# EPICS StreamDevice protocol: iocs/estherVacuumRpi/vacApp/Db/gate-valve.proto
Terminator = CR LF;
#Terminator = LF;
#LockTimeout = 5000;
ReplyTimeout = 2000;
#ReadTimeout  = 200;
#WriteTimeout = 100;
MaxInput     = 100;
#ExtraInput   = Error;
#ExtraInput   = Ignore;

#      "1, Closed, Char:x, SwIN:0, SwOUT:0, LimIN:1, LimOUT:0, Millis:1210605, Holding:1147167"

#1, Stopped, Char:x, SwIN:0, SwOUT:0, LimIN:0, LimOUT:0, Millis:686343, Holding:0
Millis {
    in "\$1, %*{Stopped|MovingIn|MovingOut|Closed|Open|Error}, Char:%*c, SwIN:%*b, SwOUT:%*b, LimIN:%*b, LimOUT:%*b, Millis:%d, Holding:%*d";
}
Box {
    in "%d, Closed, Char: x, SwIN: %*d, SwOUT: 0, LimIN: 1, LimOUT: 0, Millis: %*d,%*20c";
}
SwitchIn {
    in "\$1, %*{Stopped|MovingIn|MovingOut|Closed|Open|Error}, Char:%*c, SwIN:%b, SwOUT:%*b, LimIN:%*b, LimOUT:%*b, Millis:%*d, Holding:%*d";
}
SwitchInCmd {
    out "%{x|i|I}"
}

SwitchOut {
    in "\$1, %*{Stopped|MovingIn|MovingOut|Closed|Open|Error}, Char:%*c, SwIN:%*b, SwOUT:%b, LimIN:%*b, LimOUT:%*b, Millis:%*d, Holding:%*d";
}

SwitchOutCmd {
    out "%{x|o|O}"
}

StopCmd {
    out "s"
}

LimitIn {
    in "\$1, %*{Stopped|MovingIn|MovingOut|Closed|Open|Error}, Char:%*c, SwIN:%*b, SwOUT:%*b, LimIN:%b, LimOUT:%*b, Millis:%*d, Holding:%*d";
}

LimitOut {
    in "\$1, %*{Stopped|MovingIn|MovingOut|Closed|Open|Error}, Char:%*c, SwIN:%*b, SwOUT:%*b, LimIN:%*b, LimOUT:%b, Millis:%*d, Holding:%*d";
}

Status {
    in "\$1, %{Stopped|MovingIn|MovingOut|Closed|Open|Error}, Char:%*c, SwIN:%*b, SwOUT:%*b, LimIN:%*b, LimOUT:%*b, Millis:%*d, Holding:%*d";
}

    #in "\$1, %*{Stopped|MovingIn|MovingOut|Closed|Open|Error}, Char:%c, SwIN:%*b, SwOUT:%*b, LimIN:%*b, LimOUT:%*b, Millis:%*d, Holding:%*d";
Char {
    in "\$1, %*{Stopped|MovingIn|MovingOut|Closed|Open|Error}, Char:%1[xIioO], SwIN:%*b, SwOUT:%*b, LimIN:%*b, LimOUT:%*b, Millis:%*d, Holding:%*d";
}

Holding {
    in "\$1, %*{Stopped|MovingIn|MovingOut|Closed|Open|Error}, Char:%*c, SwIN:%*b, SwOUT:%*b, LimIN:%*b, LimOUT:%*b, Millis:%*d, Holding:%d";
}
debug {
    ExtraInput = Ignore;
    out "%s"; in "%60c"
}
